// TIA Portal V20 export
// export: Created 2025-12-01T14:57:44.8491488Z, ExportSetting None, DisplayName Totally Integrated Automation Portal, DisplayVersion V20 Update 3, DisplayName TIA Portal Openness, DisplayVersion V20 Update 3, DisplayName TIA Portal Version Control Interface, DisplayVersion V20 Update 3, DisplayName STEP 7 Professional, DisplayVersion V20 Update 3, DisplayName STEP 7 Safety, DisplayVersion V20 Update 2, DisplayName WinCC Basic/Comfort/Advanced, DisplayVersion V20 Update 3, DisplayName WinCC Professional, DisplayVersion V20 Update 3, DisplayName WinCC Unified, DisplayVersion V20 Update 3
FUNCTION "FC717_Emision_Routing" : Void   // FC717, SCL
{ S7_Optimized_Access := 'FALSE' }
// stored: AutoNumber false, SetENOAutomatically false
   VAR_INPUT
      NumJDT : UInt;
   END_VAR
   VAR_TEMP
      i : UInt;
      posicion : Int;
      cero : Byte;
      retval : Int;
      Numero_evento : Int;
      contador : Int;
      mode : DWord;
      separador : Char;
      longitud : Int;
      ver_numero_evento : Int;
      Destino_copia : Int;
      origen_copia : Int;
   END_VAR
BEGIN
   REGION inicializacion
       // definición del modo de union de cadenas
       // 
       #mode := 0;
       #mode.%X0 := 0;
       #mode.%X3 := 0;
       #separador := ',';
       #cero := 0;
       #Destino_copia := 0;

   END_REGION

   // evaluar hacia que JDT tenemos que emitir
   IF #NumJDT = 1 THEN
       GOTO JDT_1;
   ELSE
       GOTO JDT_2;
   END_IF;


   REGION emision JDT1
   JDT_1:   // miramos si tenemos algún mensaje que emitir
       FOR #Numero_evento := 0 TO 100 BY 1 DO
           IF LEN("DB198_eventos_generados_routing_JDT1".evento[#Numero_evento]) > 0 THEN
               // tenemos un mensaje que emitir. miramos si hay espacio en la emisión
               FOR #i := 0 TO "JDT1_MaxBytes" BY 1 DO //
                   IF (("DB808_JDT01EventosGenerados".Mensaje[#i] = #cero) OR ("DB808_JDT01EventosGenerados".Mensaje[#i] = ' ')) THEN
                       #posicion := #i;
                       #ver_numero_evento := #Numero_evento;
                       GOTO Formateo_JDT1;
                   END_IF;
               END_FOR;
               //si no hemos ido a la emisión es que no hay espacio
               // aqui tenemos que reordenar los mensajes no emitidos
               REGION reordena mensajes pendientes
                   // buscamos la primera posición donde tenemos mensaje
                   FOR #origen_copia:=0 TO 100 BY 1 DO
                       IF LEN("DB198_eventos_generados_routing_JDT1".evento[#origen_copia]) > 0 THEN
                           IF #origen_copia = 0 THEN
                               // si es cero es que no hay que reordenar.
                               RETURN;
                           ELSE
                               "DB198_eventos_generados_routing_JDT1".evento[#Destino_copia] := "DB198_eventos_generados_routing_JDT1".evento[#origen_copia];
                               "DB198_eventos_generados_routing_JDT1".evento[#origen_copia] := '';
                               #Destino_copia += 1;
                           END_IF;
                       END_IF;
                   END_FOR;
               END_REGION
               RETURN; // despues de reordenar salimos de la función

           Formateo_JDT1:
               // si no es el primer mensaje tenemos que añadir una coma
               // 
               IF #posicion > 0 THEN
                   "DB808_JDT01EventosGenerados".Mensaje[#posicion] := ',';
                   #posicion += 1;
               END_IF;

               #retval := JOIN(Mode := #mode, RecSeparator := #separador, EndSeparator := #separador, SrcStruct := "DB198_eventos_generados_routing_JDT1".evento[#Numero_evento], Count := #contador, DstArray := "DB808_JDT01EventosGenerados".Mensaje, Position := #posicion);
               "DB198_eventos_generados_routing_JDT1".evento[#Numero_evento] := ''; //eliminamos el mensaje emitido
           END_IF;
           ;
           // primero tenemos que evaluar si hay espacio para formatear eventos
       END_FOR;
   END_REGION


   REGION emision JDT2

   JDT_2:// miramos si tenemos algún mensaje que emitir
       FOR #Numero_evento := 0 TO 100 BY 1 DO
           IF LEN("DB197_eventos_generados_routing_JDT2".evento[#Numero_evento]) > 0 THEN
               // tenemos un mensaje que emitir. miramos si hay espacio en la emisión
               FOR #i := 0 TO "JDT2_MaxBytes" BY 1 DO //
                   IF (("DB707_JDT02EventosGenerados".Mensaje[#i] = #cero) OR ("DB707_JDT02EventosGenerados".Mensaje[#i] = ' ')) THEN
                       #posicion := #i;
                       #ver_numero_evento := #Numero_evento;
                       GOTO Formateo_JDT2;
                   END_IF;
               END_FOR;
               //si no hemos ido a la emisión es que no hay espacio
               // aqui tenemos que reordenar los mensajes no emitidos
               REGION reordena mensajes pendientes
                   // buscamos la primera posición donde tenemos mensaje
                   FOR #origen_copia := 0 TO 100 BY 1 DO
                       IF LEN("DB197_eventos_generados_routing_JDT2".evento[#origen_copia]) > 0 THEN
                           IF #origen_copia = 0 THEN
                               // si es cero es que no hay que reordenar.
                               RETURN;
                           ELSE
                               "DB197_eventos_generados_routing_JDT2".evento[#Destino_copia] := "DB197_eventos_generados_routing_JDT2".evento[#origen_copia];
                               "DB197_eventos_generados_routing_JDT2".evento[#origen_copia] := '';
                               #Destino_copia += 1;
                           END_IF;
                       END_IF;
                   END_FOR;
               END_REGION
               RETURN; // despues de reordenar salimos de la función

           Formateo_JDT2:
               // si no es el primer mensaje tenemos que añadir una coma
               // 
               IF #posicion > 0 THEN
                   "DB707_JDT02EventosGenerados".Mensaje[#posicion] := ',';
                   #posicion += 1;
               END_IF;
               #retval := JOIN(Mode := #mode, RecSeparator := #separador, EndSeparator := #separador, SrcStruct := "DB197_eventos_generados_routing_JDT2".evento[#Numero_evento], Count := #contador, DstArray := "DB707_JDT02EventosGenerados".Mensaje, Position := #posicion);
               "DB197_eventos_generados_routing_JDT2".evento[#Numero_evento] := ''; //eliminamos el mensaje emitido
           END_IF;
           ;
           // primero tenemos que evaluar si hay espacio para formatear eventos
       END_FOR;
   END_REGION
END_FUNCTION
